(* Logix 5000 project; controller DispersionPlc vendor 1 type 14 code 108 rev 34.11; software revision 34.01; part 19 of 22 *)
(* tags used below, declared in another part *)
   Cool_SP : REAL;
   Cool_SP2 : REAL;
   Cool_SP3 : REAL;
   DummyOutput : BOOL;
   Estop_Disp : ALIAS FOR Local:3:I.Data.1;
   FIT_4305_xx : AStd_AnalogInput;
   Heat_SP : REAL;
   LS_4302_High : BOOL;
   Normal_SP : REAL;
   PCV_4302_3 : AStd_VlvModulating;
   PIC_4302_3 : AStd_PIDInterface;
   PIC_4302_3_AOI : AStd_PIDInterface_AOI;
   PIC_4302_3_Mode : SINT;
   PIC_4302_3_PID : PID_ENHANCED;
   PIC_4302_3_Setpoint : REAL;
   PIT_4302_2 : AStd_AnalogInput;
   RO_HE4305_PhaseROWaterAddition : AStd_PLI;
   SPARE_I414 : ALIAS FOR Local:4:I.Data.14;
   SPARE_O714 : ALIAS FOR Local:7:O.Data.14;
   SV_4306_1 : AStd_VlvOC;
   SV_4306_1_AOI : AStd_VlvOC_AOI;
   T4302_PhaseTempControl : AStd_PLI;
   TC_4305_1 : AStd_PIDInterface;
   TIT_4302_4 : AStd_AnalogInput;
   TIT_4305_1 : AStd_AnalogInput;
   TIT_4306_1 : AStd_AnalogInput;
   TIT_4306_1_AOI : AStd_AI_AOI;
   VFD_4306_1 : AStd_VFD;
   VFD_4306_1_AOI : AStd_VFD_AOI;
   WIT_4302_1 : AStd_AnalogInput;
   WIT_4306_1 : AStd_AnalogInput;
   WIT_4306_1_AOI : AStd_AI_AOI;
   XV_4301_8 : AStd_VlvOC;
   XV_4302_10 : AStd_VlvOC;
   XV_4302_8 : AStd_VlvOC;
   XV_4306_1 : AStd_VlvOC;
   XV_4306_1_AOI : AStd_VlvOC_AOI;
   XV_4306_1_IOpn : BOOL;
   XV_4306_1_OCls : BOOL;
   XV_4306_2 : AStd_VlvOC;
   XV_4306_2_AOI : AStd_VlvOC_AOI;
   XV_4306_2_IOpn : BOOL;
   XV_4306_2_OCls : BOOL;
   XV_4306_3 : AStd_VlvOC;
   XV_4306_3_AOI : AStd_VlvOC_AOI;
   XV_4306_3_IOpn : BOOL;
   XV_4306_3_OCls : BOOL;
   XV_4306_4 : AStd_VlvOC;
   XV_4306_4_AOI : AStd_VlvOC_AOI;
   XV_4306_4_IOpn : BOOL;
   XV_4306_4_OCls : BOOL;
   XV_4306_5 : AStd_VlvOC;
   XV_4306_5_AOI : AStd_VlvOC_AOI;
   XV_4306_5_IOpn : BOOL;
   XV_4306_5_OCls : BOOL;
   XV_4307_3 : AStd_VlvOC;
   XV_4307_6 : AStd_VlvOC;
(* Unit_T4302, continued *)

ROUTINE PIC_4302_3   (* ladder *)
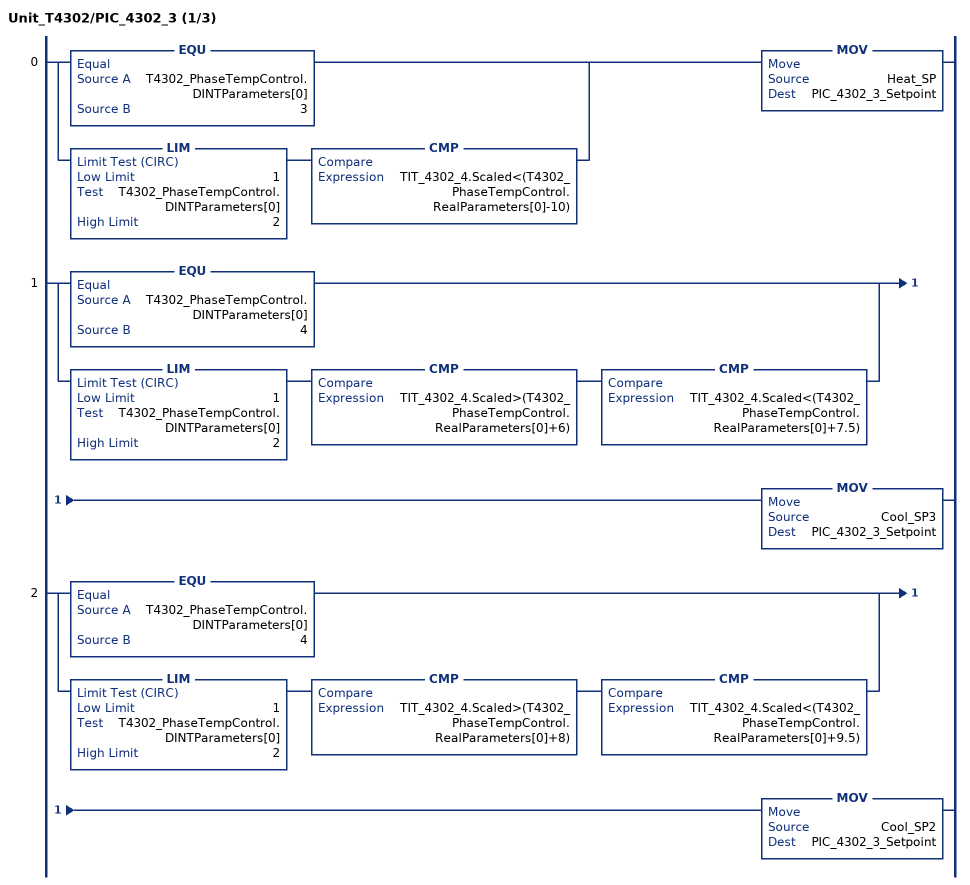
   0: [EQU(T4302_PhaseTempControl.DINTParameters[0],3) ,LIM(1,T4302_PhaseTempControl.DINTParameters[0],2) CMP(TIT_4302_4.Scaled<(T4302_PhaseTempControl.RealParameters[0]-10)) ]MOV(Heat_SP,PIC_4302_3_Setpoint);
   1: [EQU(T4302_PhaseTempControl.DINTParameters[0],4) ,LIM(1,T4302_PhaseTempControl.DINTParameters[0],2) CMP(TIT_4302_4.Scaled>(T4302_PhaseTempControl.RealParameters[0]+6)) CMP(TIT_4302_4.Scaled<(T4302_PhaseTempControl.RealParameters[0]+7.5)) ]MOV(Cool_SP3,PIC_4302_3_Setpoint);
   2: [EQU(T4302_PhaseTempControl.DINTParameters[0],4) ,LIM(1,T4302_PhaseTempControl.DINTParameters[0],2) CMP(TIT_4302_4.Scaled>(T4302_PhaseTempControl.RealParameters[0]+8)) CMP(TIT_4302_4.Scaled<(T4302_PhaseTempControl.RealParameters[0]+9.5)) ]MOV(Cool_SP2,PIC_4302_3_Setpoint);
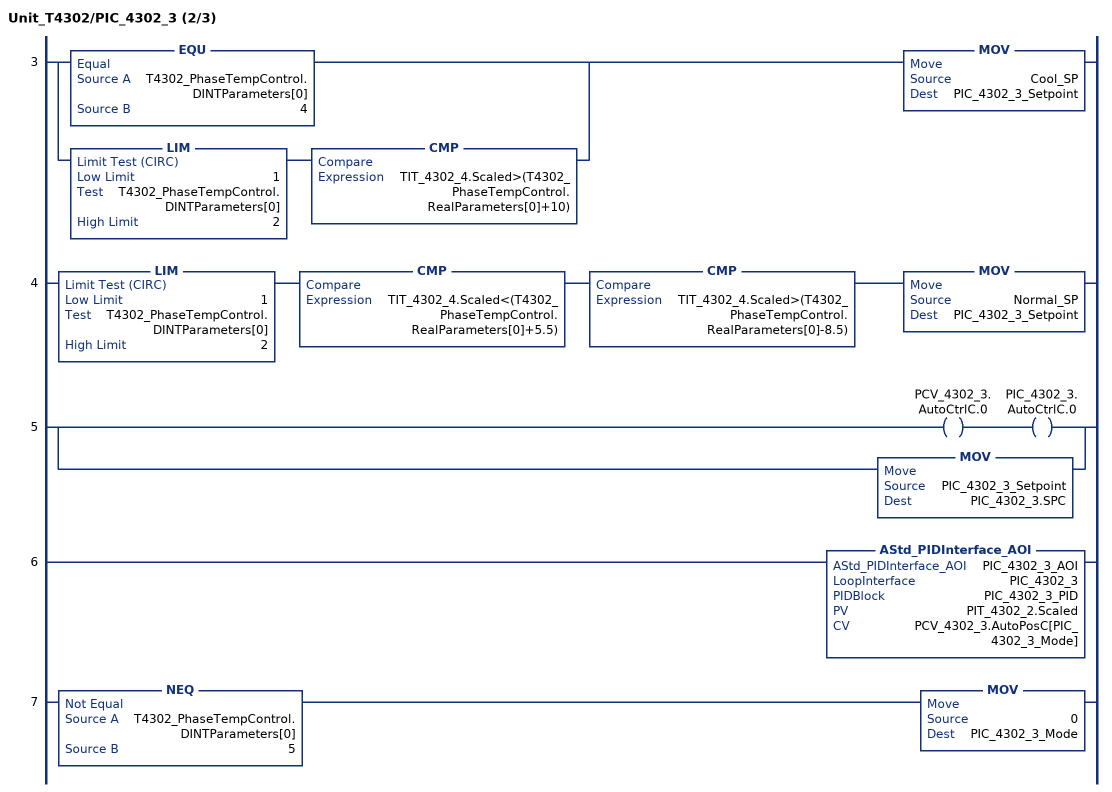
   3: [EQU(T4302_PhaseTempControl.DINTParameters[0],4) ,LIM(1,T4302_PhaseTempControl.DINTParameters[0],2) CMP(TIT_4302_4.Scaled>(T4302_PhaseTempControl.RealParameters[0]+10)) ]MOV(Cool_SP,PIC_4302_3_Setpoint);
   4: LIM(1,T4302_PhaseTempControl.DINTParameters[0],2)CMP(TIT_4302_4.Scaled<(T4302_PhaseTempControl.RealParameters[0]+5.5))CMP(TIT_4302_4.Scaled>(T4302_PhaseTempControl.RealParameters[0]-8.5))MOV(Normal_SP,PIC_4302_3_Setpoint);
   5: [OTE(PCV_4302_3.AutoCtrlC.0) OTE(PIC_4302_3.AutoCtrlC.0) ,MOV(PIC_4302_3_Setpoint,PIC_4302_3.SPC) ];
   6: AStd_PIDInterface_AOI(PIC_4302_3_AOI,PIC_4302_3,PIC_4302_3_PID,PIT_4302_2.Scaled,PCV_4302_3.AutoPosC[PIC_4302_3_Mode]);
   7: NEQ(T4302_PhaseTempControl.DINTParameters[0],5)MOV(0,PIC_4302_3_Mode);
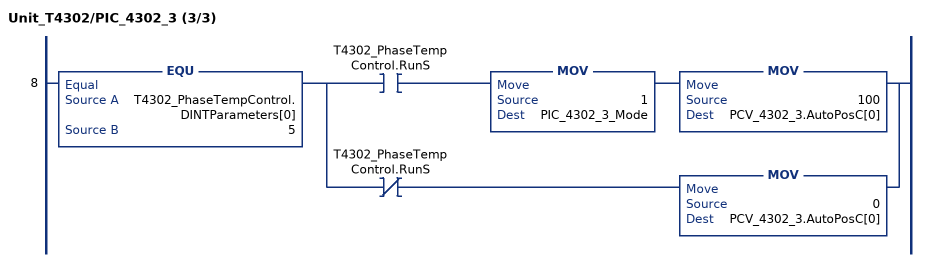
   8: EQU(T4302_PhaseTempControl.DINTParameters[0],5)[XIC(T4302_PhaseTempControl.RunS) MOV(1,PIC_4302_3_Mode) MOV(100,PCV_4302_3.AutoPosC[0]) ,XIO(T4302_PhaseTempControl.RunS) MOV(0,PCV_4302_3.AutoPosC[0]) ];
END_ROUTINE
END_PROGRAM

PROGRAM Unit_V4306   (* main routine MainRoutine *)

ROUTINE Device_SV_4306_1   (* ladder *)
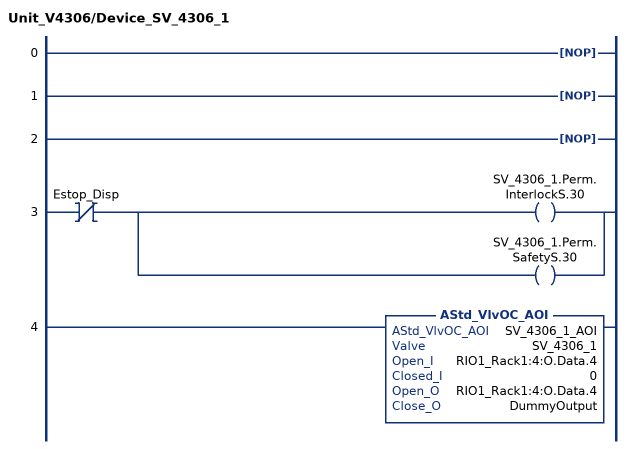
   0: NOP();
   1: NOP();
   2: NOP();
   3: XIO(Estop_Disp)[OTE(SV_4306_1.Perm.InterlockS.30) ,OTE(SV_4306_1.Perm.SafetyS.30) ];
   4: AStd_VlvOC_AOI(SV_4306_1_AOI,SV_4306_1,RIO1_Rack1:4:O.Data.4,0,RIO1_Rack1:4:O.Data.4,DummyOutput);
END_ROUTINE

ROUTINE Device_TIC_4305_1   (* ladder *)
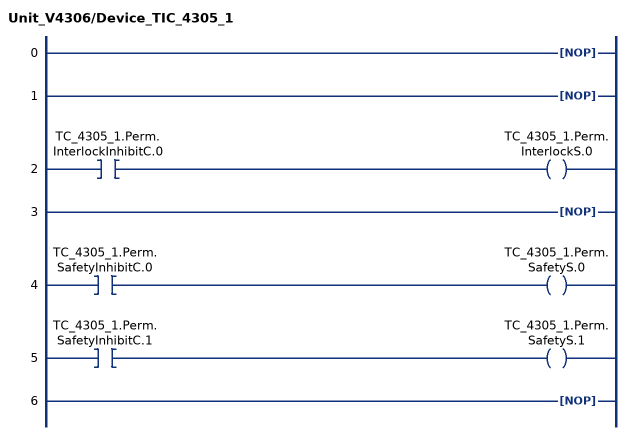
   0: NOP();
   1: NOP();
   2: XIC(TC_4305_1.Perm.InterlockInhibitC.0)OTE(TC_4305_1.Perm.InterlockS.0);
   3: NOP();
   4: XIC(TC_4305_1.Perm.SafetyInhibitC.0)OTE(TC_4305_1.Perm.SafetyS.0);
   5: XIC(TC_4305_1.Perm.SafetyInhibitC.1)OTE(TC_4305_1.Perm.SafetyS.1);
   6: NOP();
END_ROUTINE

ROUTINE Device_TIT_4306_1   (* ladder *)
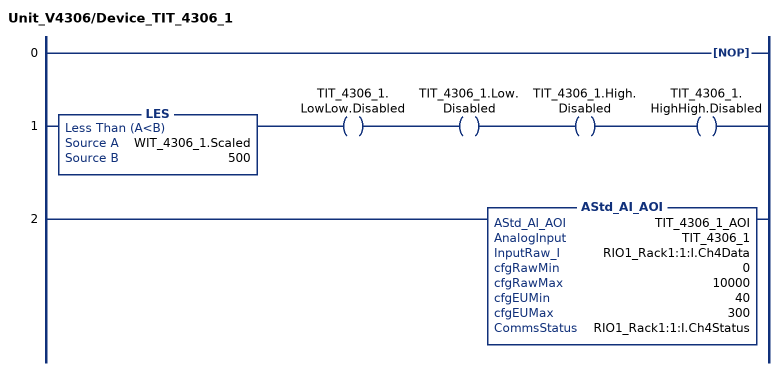
   0: NOP();
   1: LES(WIT_4306_1.Scaled,500)OTE(TIT_4306_1.LowLow.Disabled)OTE(TIT_4306_1.Low.Disabled)OTE(TIT_4306_1.High.Disabled)OTE(TIT_4306_1.HighHigh.Disabled);
   2: AStd_AI_AOI(TIT_4306_1_AOI,TIT_4306_1,RIO1_Rack1:1:I.Ch4Data,0,10000,40,300,RIO1_Rack1:1:I.Ch4Status);
END_ROUTINE

ROUTINE Device_VFD_4306_1   (* ladder *)
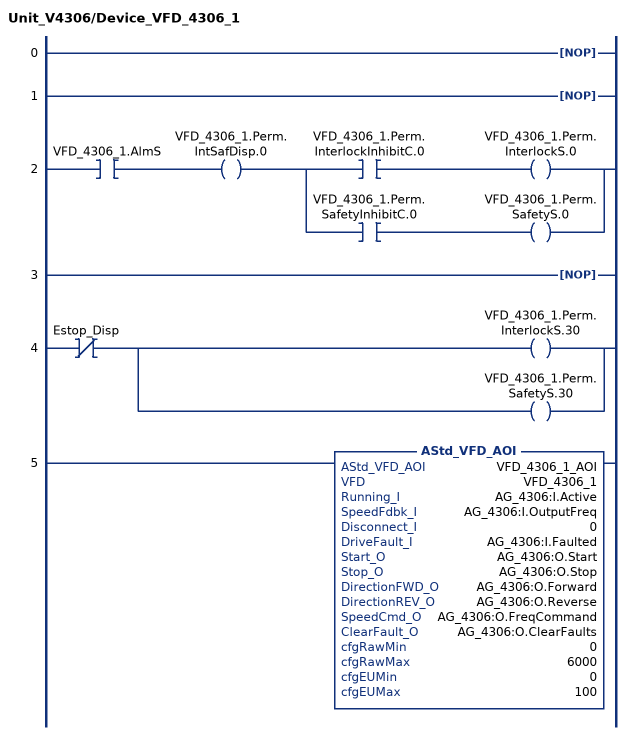
   0: NOP();
   1: NOP();
   2: XIC(VFD_4306_1.AlmS)OTE(VFD_4306_1.Perm.IntSafDisp.0)[XIC(VFD_4306_1.Perm.InterlockInhibitC.0) OTE(VFD_4306_1.Perm.InterlockS.0) ,XIC(VFD_4306_1.Perm.SafetyInhibitC.0) OTE(VFD_4306_1.Perm.SafetyS.0) ];
   3: NOP();
   4: XIO(Estop_Disp)[OTE(VFD_4306_1.Perm.InterlockS.30) ,OTE(VFD_4306_1.Perm.SafetyS.30) ];
   5: AStd_VFD_AOI(VFD_4306_1_AOI,VFD_4306_1,AG_4306:I.Active,AG_4306:I.OutputFreq,0,AG_4306:I.Faulted,AG_4306:O.Start,AG_4306:O.Stop,AG_4306:O.Forward,AG_4306:O.Reverse,AG_4306:O.FreqCommand,AG_4306:O.ClearFaults,0,6000,0,100);
END_ROUTINE

ROUTINE Device_WIT_4306_1   (* ladder *)
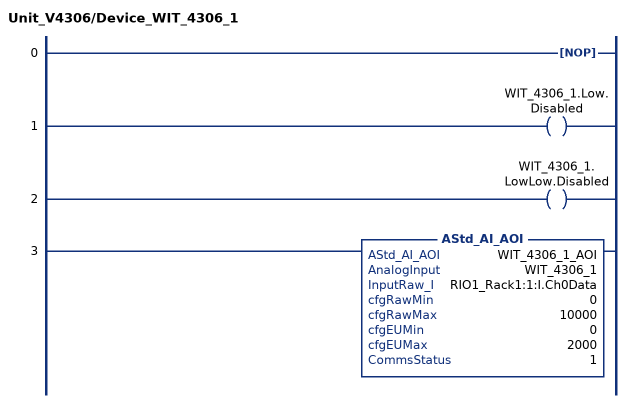
   0: NOP();
   1: OTE(WIT_4306_1.Low.Disabled);
   2: OTE(WIT_4306_1.LowLow.Disabled);
   3: AStd_AI_AOI(WIT_4306_1_AOI,WIT_4306_1,RIO1_Rack1:1:I.Ch0Data,0,10000,0,2000,1);
END_ROUTINE

ROUTINE Device_XV_4306_1   (* ladder *)
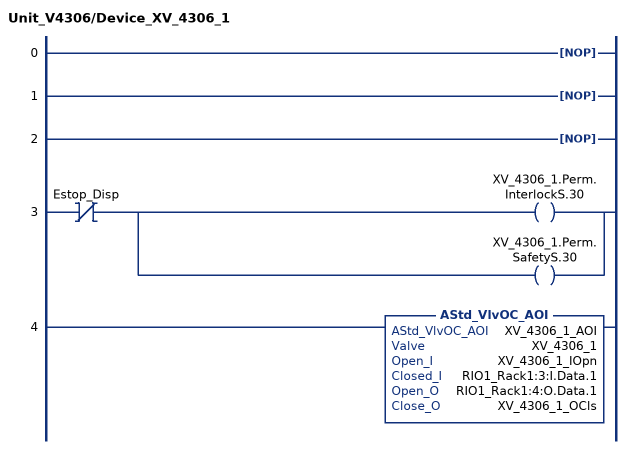
   0: NOP();
   1: NOP();
   2: NOP();
   3: XIO(Estop_Disp)[OTE(XV_4306_1.Perm.InterlockS.30) ,OTE(XV_4306_1.Perm.SafetyS.30) ];
   4: AStd_VlvOC_AOI(XV_4306_1_AOI,XV_4306_1,XV_4306_1_IOpn,RIO1_Rack1:3:I.Data.1,RIO1_Rack1:4:O.Data.1,XV_4306_1_OCls);
END_ROUTINE

ROUTINE Device_XV_4306_2   (* ladder *)
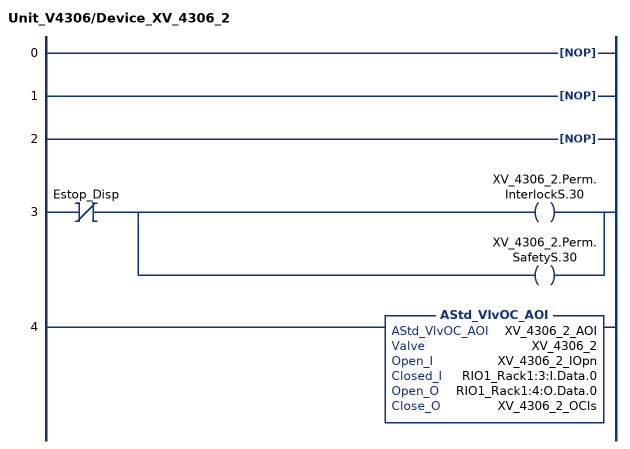
   0: NOP();
   1: NOP();
   2: NOP();
   3: XIO(Estop_Disp)[OTE(XV_4306_2.Perm.InterlockS.30) ,OTE(XV_4306_2.Perm.SafetyS.30) ];
   4: AStd_VlvOC_AOI(XV_4306_2_AOI,XV_4306_2,XV_4306_2_IOpn,RIO1_Rack1:3:I.Data.0,RIO1_Rack1:4:O.Data.0,XV_4306_2_OCls);
END_ROUTINE

ROUTINE Device_XV_4306_3   (* ladder *)
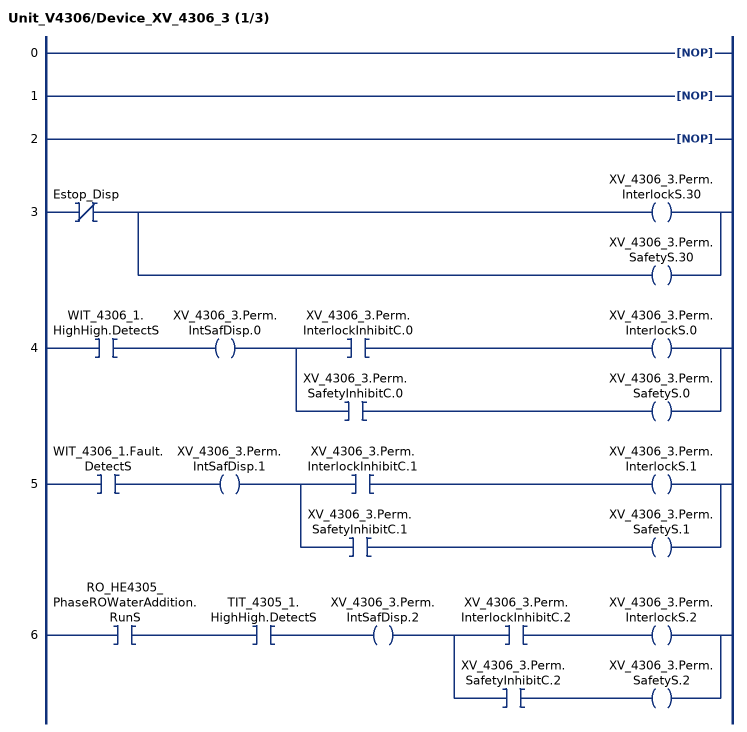
   0: NOP();
   1: NOP();
   2: NOP();
   3: XIO(Estop_Disp)[OTE(XV_4306_3.Perm.InterlockS.30) ,OTE(XV_4306_3.Perm.SafetyS.30) ];
   4: XIC(WIT_4306_1.HighHigh.DetectS)OTE(XV_4306_3.Perm.IntSafDisp.0)[XIC(XV_4306_3.Perm.InterlockInhibitC.0) OTE(XV_4306_3.Perm.InterlockS.0) ,XIC(XV_4306_3.Perm.SafetyInhibitC.0) OTE(XV_4306_3.Perm.SafetyS.0) ];
   5: XIC(WIT_4306_1.Fault.DetectS)OTE(XV_4306_3.Perm.IntSafDisp.1)[XIC(XV_4306_3.Perm.InterlockInhibitC.1) OTE(XV_4306_3.Perm.InterlockS.1) ,XIC(XV_4306_3.Perm.SafetyInhibitC.1) OTE(XV_4306_3.Perm.SafetyS.1) ];
   6: XIC(RO_HE4305_PhaseROWaterAddition.RunS)XIC(TIT_4305_1.HighHigh.DetectS)OTE(XV_4306_3.Perm.IntSafDisp.2)[XIC(XV_4306_3.Perm.InterlockInhibitC.2) OTE(XV_4306_3.Perm.InterlockS.2) ,XIC(XV_4306_3.Perm.SafetyInhibitC.2) OTE(XV_4306_3.Perm.SafetyS.2) ];
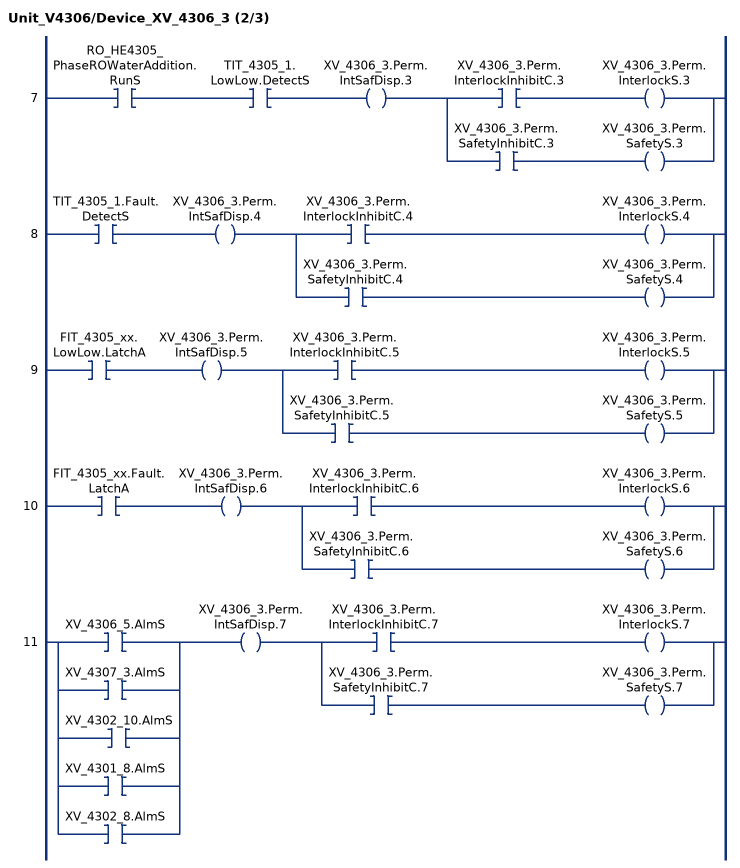
   7: XIC(RO_HE4305_PhaseROWaterAddition.RunS)XIC(TIT_4305_1.LowLow.DetectS)OTE(XV_4306_3.Perm.IntSafDisp.3)[XIC(XV_4306_3.Perm.InterlockInhibitC.3) OTE(XV_4306_3.Perm.InterlockS.3) ,XIC(XV_4306_3.Perm.SafetyInhibitC.3) OTE(XV_4306_3.Perm.SafetyS.3) ];
   8: XIC(TIT_4305_1.Fault.DetectS)OTE(XV_4306_3.Perm.IntSafDisp.4)[XIC(XV_4306_3.Perm.InterlockInhibitC.4) OTE(XV_4306_3.Perm.InterlockS.4) ,XIC(XV_4306_3.Perm.SafetyInhibitC.4) OTE(XV_4306_3.Perm.SafetyS.4) ];
   9: XIC(FIT_4305_xx.LowLow.LatchA)OTE(XV_4306_3.Perm.IntSafDisp.5)[XIC(XV_4306_3.Perm.InterlockInhibitC.5) OTE(XV_4306_3.Perm.InterlockS.5) ,XIC(XV_4306_3.Perm.SafetyInhibitC.5) OTE(XV_4306_3.Perm.SafetyS.5) ];
   10: XIC(FIT_4305_xx.Fault.LatchA)OTE(XV_4306_3.Perm.IntSafDisp.6)[XIC(XV_4306_3.Perm.InterlockInhibitC.6) OTE(XV_4306_3.Perm.InterlockS.6) ,XIC(XV_4306_3.Perm.SafetyInhibitC.6) OTE(XV_4306_3.Perm.SafetyS.6) ];
   11: [XIC(XV_4306_5.AlmS) ,XIC(XV_4307_3.AlmS) ,XIC(XV_4302_10.AlmS) ,XIC(XV_4301_8.AlmS) ,XIC(XV_4302_8.AlmS) ]OTE(XV_4306_3.Perm.IntSafDisp.7)[XIC(XV_4306_3.Perm.InterlockInhibitC.7) OTE(XV_4306_3.Perm.InterlockS.7) ,XIC(XV_4306_3.Perm.SafetyInhibitC.7) OTE(XV_4306_3.Perm.SafetyS.7) ];
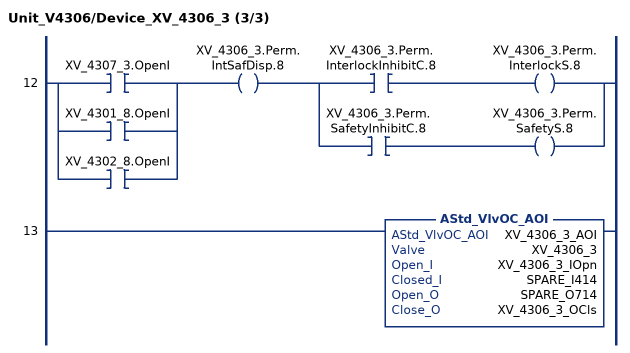
   12: [XIC(XV_4307_3.OpenI) ,XIC(XV_4301_8.OpenI) ,XIC(XV_4302_8.OpenI) ]OTE(XV_4306_3.Perm.IntSafDisp.8)[XIC(XV_4306_3.Perm.InterlockInhibitC.8) OTE(XV_4306_3.Perm.InterlockS.8) ,XIC(XV_4306_3.Perm.SafetyInhibitC.8) OTE(XV_4306_3.Perm.SafetyS.8) ];
   13: AStd_VlvOC_AOI(XV_4306_3_AOI,XV_4306_3,XV_4306_3_IOpn,SPARE_I414,SPARE_O714,XV_4306_3_OCls);
END_ROUTINE

ROUTINE Device_XV_4306_4   (* ladder *)
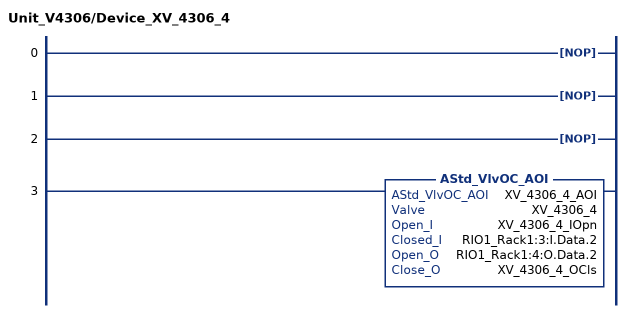
   0: NOP();
   1: NOP();
   2: NOP();
   3: AStd_VlvOC_AOI(XV_4306_4_AOI,XV_4306_4,XV_4306_4_IOpn,RIO1_Rack1:3:I.Data.2,RIO1_Rack1:4:O.Data.2,XV_4306_4_OCls);
END_ROUTINE

ROUTINE Device_XV_4306_5   (* ladder *)
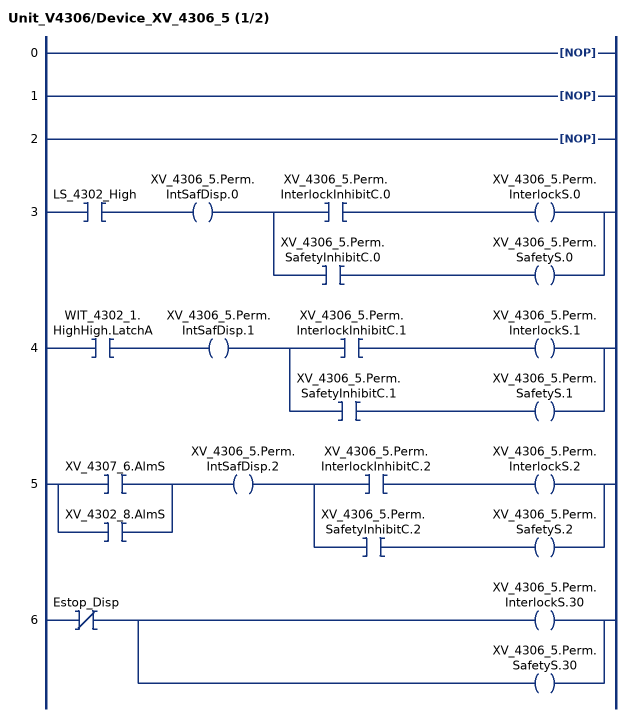
   0: NOP();
   1: NOP();
   2: NOP();
   3: XIC(LS_4302_High)OTE(XV_4306_5.Perm.IntSafDisp.0)[XIC(XV_4306_5.Perm.InterlockInhibitC.0) OTE(XV_4306_5.Perm.InterlockS.0) ,XIC(XV_4306_5.Perm.SafetyInhibitC.0) OTE(XV_4306_5.Perm.SafetyS.0) ];
   4: XIC(WIT_4302_1.HighHigh.LatchA)OTE(XV_4306_5.Perm.IntSafDisp.1)[XIC(XV_4306_5.Perm.InterlockInhibitC.1) OTE(XV_4306_5.Perm.InterlockS.1) ,XIC(XV_4306_5.Perm.SafetyInhibitC.1) OTE(XV_4306_5.Perm.SafetyS.1) ];
   5: [XIC(XV_4307_6.AlmS) ,XIC(XV_4302_8.AlmS) ]OTE(XV_4306_5.Perm.IntSafDisp.2)[XIC(XV_4306_5.Perm.InterlockInhibitC.2) OTE(XV_4306_5.Perm.InterlockS.2) ,XIC(XV_4306_5.Perm.SafetyInhibitC.2) OTE(XV_4306_5.Perm.SafetyS.2) ];
   6: XIO(Estop_Disp)[OTE(XV_4306_5.Perm.InterlockS.30) ,OTE(XV_4306_5.Perm.SafetyS.30) ];
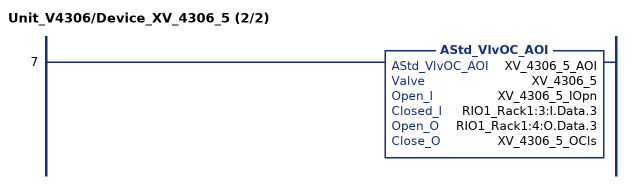
   7: AStd_VlvOC_AOI(XV_4306_5_AOI,XV_4306_5,XV_4306_5_IOpn,RIO1_Rack1:3:I.Data.3,RIO1_Rack1:4:O.Data.3,XV_4306_5_OCls);
END_ROUTINE

ROUTINE MainRoutine   (* ladder *)
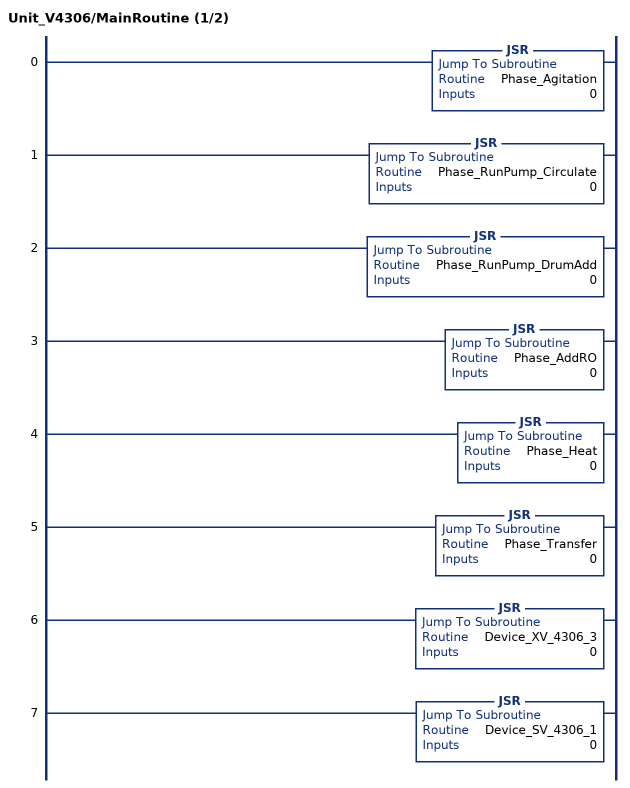
   0: JSR(Phase_Agitation,0);
   1: JSR(Phase_RunPump_Circulate,0);
   2: JSR(Phase_RunPump_DrumAdd,0);
   3: JSR(Phase_AddRO,0);
   4: JSR(Phase_Heat,0);
   5: JSR(Phase_Transfer,0);
   6: JSR(Device_XV_4306_3,0);
   7: JSR(Device_SV_4306_1,0);
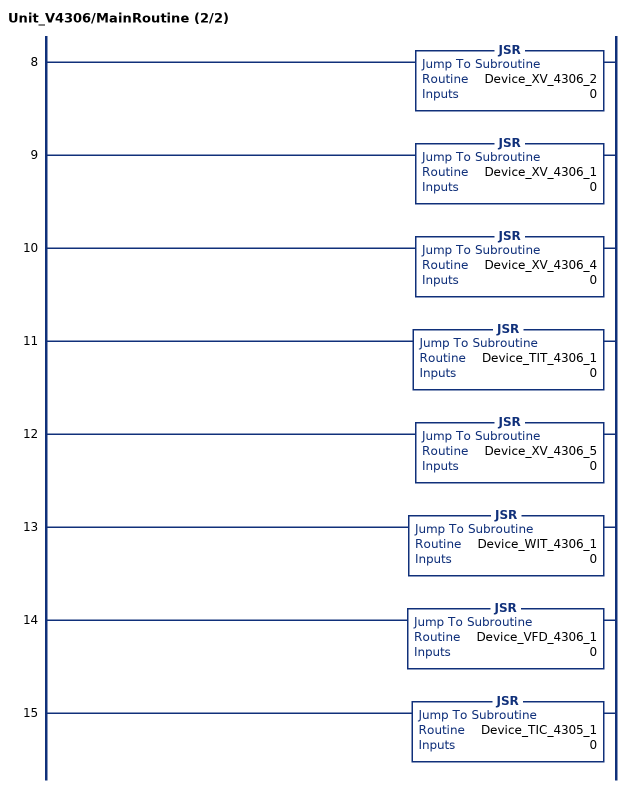
   8: JSR(Device_XV_4306_2,0);
   9: JSR(Device_XV_4306_1,0);
   10: JSR(Device_XV_4306_4,0);
   11: JSR(Device_TIT_4306_1,0);
   12: JSR(Device_XV_4306_5,0);
   13: JSR(Device_WIT_4306_1,0);
   14: JSR(Device_VFD_4306_1,0);
   15: JSR(Device_TIC_4305_1,0);
END_ROUTINE
